INTERFACE IPAScaleVolumetric EXTENDS IPAScale

END_INTERFACE

(* stored: Version 1.1.0.1, ProductVersion 3.1.4020.12
   Itf IPAScaleVolumetric: Id {c237a463-a173-43cf-bbd1-2816a810706e} *)
